# EPICS substitutions: iocBoot/ioc-tst-05/ioc-tst-05.substitutions
# IOC archive file
## Replace TST:R40:IOC:22 with the PV prefix used for
## iocAdmin PV's on this IOC

# Generate IOC archive request
file archive_ipimbIoc.archive
{
	{ IOC = "TST:R40:IOC:22" }
}
